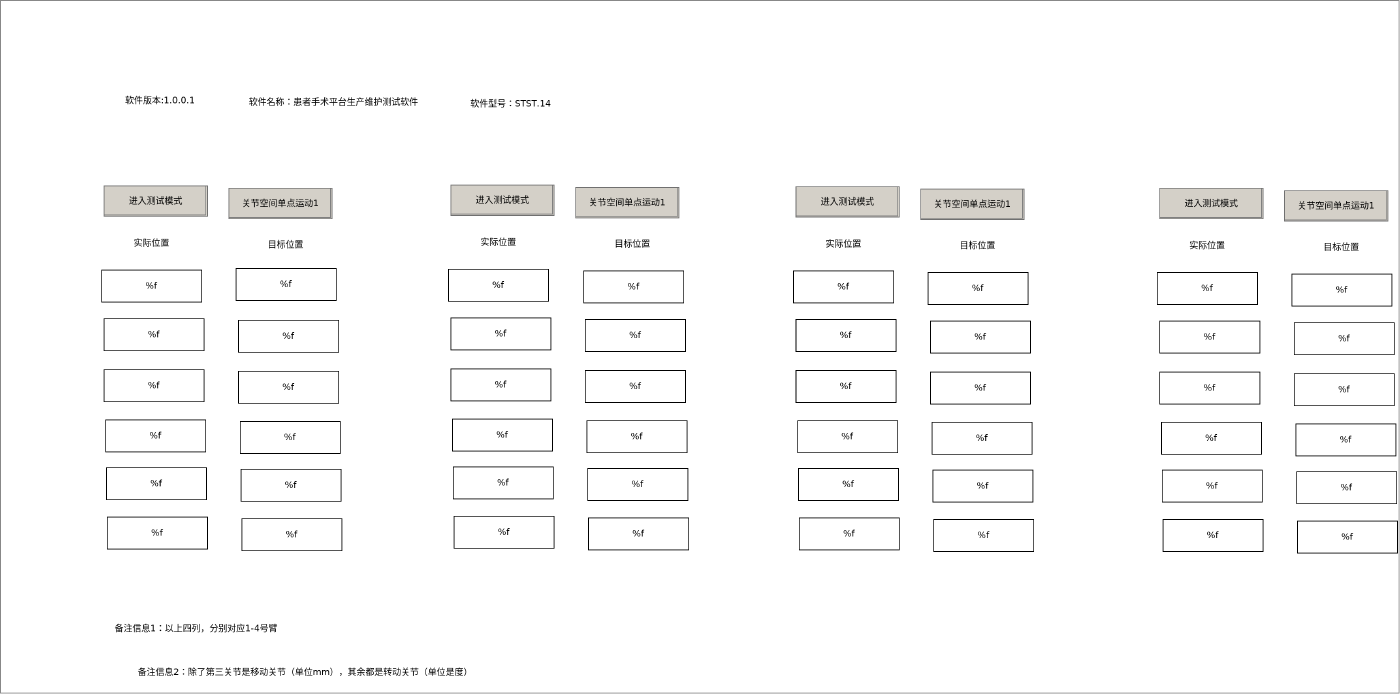
VISUALIZATION slaveArmJntTest  // 1728x857
    Button (282,232 128x38), "关节空间单点运动1", colour toggle: g_motionTest.m_uiArmModeL[1,1]
        tap g_motionTest.m_uiArmMode[1,1]
    Button (128,229 128x38), "进入测试模式", colour toggle: g_motionTest.m_enterPrecisionTestMode[1]
        toggle g_motionTest.m_enterPrecisionTestMode[1]
    Rectangle (294,395 124x40), "%f", text variable: g_motionTest.m_targetJntPos[1][2]
        OnMouseClick: write the text variable via Default
    Rectangle (294,458 124x40), "%f", text variable: g_motionTest.m_targetJntPos[1][3]
        OnMouseClick: write the text variable via Default
    Rectangle (298,640 124x40), "%f", text variable: g_motionTest.m_targetJntPos[1][6]
        OnMouseClick: write the text variable via Default
    Rectangle (296,520 124x40), "%f", text variable: g_motionTest.m_targetJntPos[1][4]
        OnMouseClick: write the text variable via Default
    Rectangle (297,579 124x40), "%f", text variable: g_motionTest.m_targetJntPos[1][5]
        OnMouseClick: write the text variable via Default
    Label (280,288 145x28), "目标位置"
    Label (112,285 150x30), "实际位置"
    Rectangle (125,333 124x40), "%f", text variable: g_motionTest.m_actDHJntPos[1][1]
    Rectangle (128,393 124x40), "%f", text variable: g_motionTest.m_actDHJntPos[1][2]
    Rectangle (128,456 124x40), "%f", text variable: g_motionTest.m_actDHJntPos[1][3]
    Rectangle (132,638 124x40), "%f", text variable: g_motionTest.m_actDHJntPos[1][6]
    Rectangle (130,518 124x40), "%f", text variable: g_motionTest.m_actDHJntPos[1][4]
    Rectangle (131,577 124x40), "%f", text variable: g_motionTest.m_actDHJntPos[1][5]
    Button (710,231 128x38), "关节空间单点运动1", colour toggle: g_motionTest.m_uiArmModeL[2,1]
        tap g_motionTest.m_uiArmMode[2,1]
    Button (556,228 128x38), "进入测试模式", colour toggle: g_motionTest.m_enterPrecisionTestMode[2]
        toggle g_motionTest.m_enterPrecisionTestMode[2]
    Rectangle (720,334 124x40), "%f", text variable: g_motionTest.m_targetJntPos[2][1]
        OnMouseClick: write the text variable via Default
    Rectangle (722,394 124x40), "%f", text variable: g_motionTest.m_targetJntPos[2][2]
        OnMouseClick: write the text variable via Default
    Rectangle (722,457 124x40), "%f", text variable: g_motionTest.m_targetJntPos[2][3]
        OnMouseClick: write the text variable via Default
    Rectangle (726,639 124x40), "%f", text variable: g_motionTest.m_targetJntPos[2][6]
        OnMouseClick: write the text variable via Default
    Rectangle (724,519 124x40), "%f", text variable: g_motionTest.m_targetJntPos[2][4]
        OnMouseClick: write the text variable via Default
    Rectangle (725,578 124x40), "%f", text variable: g_motionTest.m_targetJntPos[2][5]
        OnMouseClick: write the text variable via Default
    Label (708,287 145x28), "目标位置"
    Label (540,284 150x30), "实际位置"
    Rectangle (553,332 124x40), "%f", text variable: g_motionTest.m_actDHJntPos[2][1]
    Rectangle (556,392 124x40), "%f", text variable: g_motionTest.m_actDHJntPos[2][2]
    Rectangle (556,455 124x40), "%f", text variable: g_motionTest.m_actDHJntPos[2][3]
    Rectangle (560,637 124x40), "%f", text variable: g_motionTest.m_actDHJntPos[2][6]
    Rectangle (558,517 124x40), "%f", text variable: g_motionTest.m_actDHJntPos[2][4]
    Rectangle (559,576 124x40), "%f", text variable: g_motionTest.m_actDHJntPos[2][5]
    Button (1136,233 128x38), "关节空间单点运动1", colour toggle: g_motionTest.m_uiArmModeL[3,1]
        tap g_motionTest.m_uiArmMode[3,1]
    Button (982,230 128x38), "进入测试模式", colour toggle: g_motionTest.m_enterPrecisionTestMode[3]
        toggle g_motionTest.m_enterPrecisionTestMode[3]
    Rectangle (1145,336 124x40), "%f", text variable: g_motionTest.m_targetJntPos[3][1]
        OnMouseClick: write the text variable via Default
    Rectangle (1148,396 124x40), "%f", text variable: g_motionTest.m_targetJntPos[3][2]
        OnMouseClick: write the text variable via Default
    Rectangle (1148,459 124x40), "%f", text variable: g_motionTest.m_targetJntPos[3][3]
        OnMouseClick: write the text variable via Default
    Rectangle (1152,641 124x40), "%f", text variable: g_motionTest.m_targetJntPos[3][6]
        OnMouseClick: write the text variable via Default
    Rectangle (1150,521 124x40), "%f", text variable: g_motionTest.m_targetJntPos[3][4]
        OnMouseClick: write the text variable via Default
    Rectangle (1151,580 124x40), "%f", text variable: g_motionTest.m_targetJntPos[3][5]
        OnMouseClick: write the text variable via Default
    Label (1134,289 145x28), "目标位置"
    Label (966,286 150x30), "实际位置"
    Rectangle (979,334 124x40), "%f", text variable: g_motionTest.m_actDHJntPos[3][1]
    Rectangle (982,394 124x40), "%f", text variable: g_motionTest.m_actDHJntPos[3][2]
    Rectangle (982,457 124x40), "%f", text variable: g_motionTest.m_actDHJntPos[3][3]
    Rectangle (986,639 124x40), "%f", text variable: g_motionTest.m_actDHJntPos[3][6]
    Rectangle (984,519 124x40), "%f", text variable: g_motionTest.m_actDHJntPos[3][4]
    Rectangle (985,578 124x40), "%f", text variable: g_motionTest.m_actDHJntPos[3][5]
    Button (1585,235 128x38), "关节空间单点运动1", colour toggle: g_motionTest.m_uiArmModeL[4,1]
        tap g_motionTest.m_uiArmMode[4,1]
    Button (1431,232 128x38), "进入测试模式", colour toggle: g_motionTest.m_enterPrecisionTestMode[4]
        toggle g_motionTest.m_enterPrecisionTestMode[4]
    Rectangle (1594,338 124x40), "%f", text variable: g_motionTest.m_targetJntPos[4][1]
        OnMouseClick: write the text variable via Default
    Rectangle (1597,398 124x40), "%f", text variable: g_motionTest.m_targetJntPos[4][2]
        OnMouseClick: write the text variable via Default
    Rectangle (1597,461 124x40), "%f", text variable: g_motionTest.m_targetJntPos[4][3]
        OnMouseClick: write the text variable via Default
    Rectangle (1601,643 124x40), "%f", text variable: g_motionTest.m_targetJntPos[4][6]
        OnMouseClick: write the text variable via Default
    Rectangle (1599,523 124x40), "%f", text variable: g_motionTest.m_targetJntPos[4][4]
        OnMouseClick: write the text variable via Default
    Rectangle (1600,582 124x40), "%f", text variable: g_motionTest.m_targetJntPos[4][5]
        OnMouseClick: write the text variable via Default
    Label (1583,291 145x28), "目标位置"
    Label (1415,288 150x30), "实际位置"
    Rectangle (1428,336 124x40), "%f", text variable: g_motionTest.m_actDHJntPos[4][1]
    Rectangle (1431,396 124x40), "%f", text variable: g_motionTest.m_actDHJntPos[4][2]
    Rectangle (1431,459 124x40), "%f", text variable: g_motionTest.m_actDHJntPos[4][3]
    Rectangle (1435,641 124x40), "%f", text variable: g_motionTest.m_actDHJntPos[4][6]
    Rectangle (1433,521 124x40), "%f", text variable: g_motionTest.m_actDHJntPos[4][4]
    Rectangle (1434,580 124x40), "%f", text variable: g_motionTest.m_actDHJntPos[4][5]
    Label (87,749 310x54), "备注信息1：以上四列，分别对应1-4号臂"
    Label (51,803 651x54), "备注信息2：除了第三关节是移动关节（单位mm），其余都是转动关节（单位是度）"
    Rectangle (291,331 124x40), "%f", text variable: g_motionTest.m_targetJntPos[1][1]
        OnMouseClick: write the text variable via Default
    Label (148,96 99x56), "软件版本:1.0.0.1"
    Label (282,98 259x56), "软件名称：患者手术平台生产维护测试软件"
    Label (501,100 259x56), "软件型号：STST.14"
END_VISUALIZATION

(* stored: Version 1.1.0.1, ProductVersion 3.1.4024.11
   Visu slaveArmJntTest: Id {56a8a55e-959e-462a-baf3-6a13e4aac9d7} *)
